// TIA Portal V17 export
// export: Created 2024-08-09T12:53:15.1309504Z, ExportSetting WithDefaults, DisplayName Totally Integrated Automation Portal, DisplayVersion V17 Update 7, DisplayName TIA Portal Openness, DisplayVersion V17 Update 7, DisplayName TIA Portal Version Control Interface, DisplayVersion V17, DisplayName STEP 7 Professional, DisplayVersion V17 Update 7, DisplayName STEP 7 Safety, DisplayVersion V17 Update 6, DisplayName WinCC Professional, DisplayVersion V17 Update 7
VAR_GLOBAL   // PLC tag table "CommunCharg"
END_VAR
VAR_GLOBAL CONSTANT   // user constants
   NB_COMM : Int := 9;   // Nb maxi de commande par tournee
   NB_MAX_TOUR : Int := 4;
   MAX_COMPO_CHARG : Int := 9;
   MAX_CASE : Int := 9;
   MAX_PONT : USInt := 9;
   MAX_MOB_INCOMP : SInt := 9;   // Nb maxi de composants
   DEBCYCLE : USInt := 1;   // Bouton chargement
   DEMTARE : USInt := 2;   // Bouton chargement
   ABANDONCHARG : USInt := 3;   // Bouton chargement
   BTSUSP : USInt := 4;   // Bouton chargement
   BTAJOUT : USInt := 5;   // Bouton chargement
   BTVIDBENNE : USInt := 6;   // Bouton chargement
   BTACQPOSBENNE : USInt := 7;   // Bouton chargement
   BTARRPOSBENNE : USInt := 8;   // Bouton chargement
   BTCHGCEL : USInt := 9;   // Bouton chargement
   ARRET_OPER : Char := 'O';   // Type d'arret
   ARRET_QTE : Char := 'Q';   // Type d'arret
   ARRET_IMM : Char := 'I';   // Type d'arret
   ARRET_EVOL : Char := 'E';   // Type d'arret
   ARRET_VIDE : Char := 'V';   // Type d'arret
   ARRET_DEF : Char := 'D';   // Type d'arret
   A_COMPLETER : Char := 'C';   // Type cloture
   FIN_CHARG : Char := 'O';   // Type cloture
   _FERM : SInt := 0;   // Position Extrac
   _OUV : SInt := 1;   // Position Extrac
   _INTER : SInt := 2;   // Position Extrac
   "Boisseaux.VRAC3" : USInt := 1;   // Num du pont
   TARE : USInt := 1;
   BRUT : USInt := 2;
   Pont1 : USInt := 1;
   Pont2 : USInt := 2;
END_VAR
